Fanuc KAREL source: gmarcrg.kl

-- -----------------------------------------------------------------------
--
--   MODULE:         GMARCRG.KL
--   TITLE:          GMARCRG PROGRAM
--
--
--   WRITTEN BY:     Fanuc
--   REVISION DATE:  2016/10/08
--
--   LANGUAGE:       KAREL 8.33 R30iB
--   CONTROL GROUP:  BODY SHOP EXECUTION GROUP
--   STATUS:
--
--
--   ORDER NUMBER:   GMGBL4
--   PROJECT NAME:   GM Global Center
--
--
--         FANUC Robotics retains rights in any and all Software
--         contained in the material attached hereto and said
--         Software may not be copied or reproduced without the
--         written permission of FANUC Robotics.
--
--         All Software, (C) Copyright FANUC Robotics Corporation, 2016
--         DESCRIPTION: GM Global 4 ArcTool Register Setup
--
--
--
--         HISTORY OF CHANGES:
--
--         REVISION   DATE       BY               COMMENTS
--         --------   ---------  ---------------  --------------------
--
--
--
--
--
--------------------------------------------------------------------------
PROGRAM gmarcrg

%COMMENT = 'GM ARC REG V4.0'

%NOLOCKGROUP
%INVISIBLE
%RWACCESS
%NOPAUSE = ERROR + COMMAND + TPENABLE

%INCLUDE KLEVCCDF  -- Required for the TPERROR write command for the contants

%INCLUDE gmcfgcel  -- GM wizard variables for workcell variables that are common across all shops
%INCLUDE gmcfgerr  -- Required for the configuration for GM Error counting and logging


CONST

  Version = '2017-02-13'
  %INCLUDE gmcnstnt -- all GM constants for the wizard

VAR

  Current_Ver  IN SHADOW :STRING[32] -- Set equal to Version constant in initialization routine
  StrtinErs   : INTEGER   -- How many errors I/O error counter had when the program started
  ArcRG_Setup  IN SHADOW : BOOLEAN  -- Keeps track if routine setup arc tool register setup at least first time

ROUTINE writeLog(p_message: STRING; isError: BOOLEAN) FROM GMWIZLOG

%INCLUDE GMRDUTIL -- Utility Routine for Setting Variables
-----------------------------------------------------------------------------
ROUTINE init_arc_reg
-- PURPOSE: to initialize variables for arc register setup
--
--
-- INPUT:
--            -
-- OUTPUT:
--            -
-- CALLED BY:
--
--
-----------------------------------------------------------------------------
BEGIN



END init_arc_reg
-----------------------------------------------------------------------------
ROUTINE set_arc_reg
-- PURPOSE: set arc registers
--
--
-- INPUT:
--            -
-- OUTPUT:
--            -
-- CALLED BY:
--
--
-----------------------------------------------------------------------------
BEGIN

  Current_Ver = Version -- Set the version for reference

  IF UNINIT(ErrsInShop.ErrorsRgstrs) THEN
    ErrsInShop.ErrorsRgstrs = 0
  ENDIF
  IF UNINIT(ArcRG_Setup) OR (Reset_Cell) THEN
    ArcRG_Setup = FALSE
  ENDIF

  StrtinErs = ErrsInShop.ErrorsRgstrs -- grab current error count
  ClrUtltyErrs -- Clear all error in utility program to be used when done

  WriteLog('  Starting the Arc Register GMARCRG', FALSE)

  IF (ArcRG_Setup = TRUE) THEN -- setup has already been setup
    WriteLog('  Arc REG Already Setup', FALSE)
    IF ExecSetupAgn('Arc REGs') THEN -- ask user if they want to setup again
      ArcRG_Setup = FALSE
    ELSE
      WriteLog('  Arc REGs already Complete', FALSE)
      WriteLog('  GMARCRG Setup NOT executing again', FALSE)
      RETURN
    ENDIF
  ENDIF

  --setup routines
  init_arc_reg

  ErrsInShop.ErrorsRgstrs =  ErrsInShop.ErrorsRgstrs + (AddUtltyErrs) -- Get all errors in utility program to be added to any program errors
  IF (ErrsInShop.ErrorsRgstrs -StrtinErs) > 0 THEN -- check for I/O setup errors
    WriteLog('  Arc REGs Setup GMARCRG had ' + int2str((ErrsInShop.ErrorsRgstrs- StrtinErs))+' while executing', TRUE)
  ELSE
    WriteLog('  Arc REGs Setup completed', FALSE)
    ArcRG_Setup = TRUE
  ENDIF

  WriteLog('', FALSE)


END set_arc_reg
-----------------------------------------------------------------------------
BEGIN

END gmarcrg
